Yaskawa INFORM job: JOBSTART.JBI

/JOB
//NAME JOBSTART
//POS
///NPOS 0,0,0,0,0,0
//INST
///DATE 2018/09/03 09:27
///ATTR SC,RW,MC
NOP
DOUT OG#(75) B001
DOUT OG#(76) B002
TIMER T=0.50
DOUT OT#(578) ON
TIMER T=0.50
DOUT OT#(579) OFF
TIMER T=0.50
END
